KUKA KRL data list: CmdIface.dat

&ACCESS RVP
DEFDAT CMDIFACE PUBLIC
; ============================================================================
;  Latched copy of the command the robot is currently executing.
;
;  The interface words themselves (Robot_Cmd_*) can change under our feet at
;  any moment -- they are live network data. Everything below is a snapshot
;  taken once, at latch time, so a routine that reads Cmd_P1 halfway through
;  gets the value the command was issued with, not whatever the PLC has since
;  written.
; ============================================================================
DECL GLOBAL INT Cmd_Routine    = 0   ; routine ID being executed
DECL GLOBAL INT Cmd_P1         = 0   ; tray row, or reject selector on routine 90
DECL GLOBAL INT Cmd_P2         = 0   ; tray column
DECL GLOBAL INT Cmd_P3         = 0   ; sequence number, part A
DECL GLOBAL INT Cmd_P4         = 0   ; sequence number, part B
DECL GLOBAL INT Cmd_RetryLimit = 0   ; retries allowed before reporting faulted
DECL GLOBAL INT Cmd_Retries    = 0   ; retries consumed on this command
ENDDAT
